{attribute 'GeneratedUsingTerminal: EL3773-0000-0016'}
{attribute addProperty BoxType "EL3773-0000-0016"}
{attribute addProperty Id "L1_Voltage_StatusAT %I*L1_Voltage_Status_784F03AD8L1_Voltage_SamplesAT %I*L1_Voltage_Samples_ED678DEE20L1_Current_SamplesAT %I*L1_Current_Samples_89E078188L1_Current_Samples_1AT %I*L1_Current_Samples_3209B12F20L2_Voltage_StatusAT %I*L2_Voltage_Status_0626A0108L2_Voltage_SamplesAT %I*L2_Voltage_Samples_D91109BE20L2_Current_StatusAT %I*L2_Current_Status_F789DBA58L2_Current_SamplesAT %I*L2_Current_Samples_067F357F20L3_Voltage_StatusAT %I*L3_Voltage_Status_2C01C17B8L3_Voltage_SamplesAT %I*L3_Voltage_Samples_CAC3758E20L3_Current_StatusAT %I*L3_Current_Status_DDAEBACE8L3_Current_SamplesAT %I*L3_Current_Samples_15AD494F20AI_Timestamp_NextSync1TimeAT %I*AI_Timestamp_NextSync1Time_9AFDC2758AI_CycleCountAT %I*AI_CycleCount_B1A935A22WcStateAT %I*WcState_9091E0EB2InfoDataAT %I*InfoData_1088C70510"}
{attribute addProperty CRC "1502544242"}
{attribute addProperty Size "190"}
TYPE EL3773_598F0172 EXTENDS EtcSlaveTerminalBase_947E5A46 :
STRUCT
	{attribute addProperty Name "L1_Voltage_Status"}
	L1_Voltage_Status : L1_Voltage_Status_784F03AD;
	{attribute addProperty Name "L1_Voltage_Samples"}
	L1_Voltage_Samples : L1_Voltage_Samples_ED678DEE;
	{attribute addProperty Name "L1_Current_Samples"}
	L1_Current_Samples : L1_Current_Samples_89E07818;
	{attribute addProperty Name "L1_Current_Samples_1"}
	L1_Current_Samples_1 : L1_Current_Samples_3209B12F;
	{attribute addProperty Name "L2_Voltage_Status"}
	L2_Voltage_Status : L2_Voltage_Status_0626A010;
	{attribute addProperty Name "L2_Voltage_Samples"}
	L2_Voltage_Samples : L2_Voltage_Samples_D91109BE;
	{attribute addProperty Name "L2_Current_Status"}
	L2_Current_Status : L2_Current_Status_F789DBA5;
	{attribute addProperty Name "L2_Current_Samples"}
	L2_Current_Samples : L2_Current_Samples_067F357F;
	{attribute addProperty Name "L3_Voltage_Status"}
	L3_Voltage_Status : L3_Voltage_Status_2C01C17B;
	{attribute addProperty Name "L3_Voltage_Samples"}
	L3_Voltage_Samples : L3_Voltage_Samples_CAC3758E;
	{attribute addProperty Name "L3_Current_Status"}
	L3_Current_Status : L3_Current_Status_DDAEBACE;
	{attribute addProperty Name "L3_Current_Samples"}
	L3_Current_Samples : L3_Current_Samples_15AD494F;
	{attribute addProperty Name "AI_Timestamp_NextSync1Time"}
	AI_Timestamp_NextSync1Time : AI_Timestamp_NextSync1Time_9AFDC275;
	{attribute addProperty Name "AI_CycleCount"}
	AI_CycleCount : AI_CycleCount_B1A935A2;
	{attribute addProperty Name "WcState"}
	WcState : WcState_9091E0EB;
	{attribute addProperty Name "InfoData"}
	InfoData : InfoData_1088C705;
END_STRUCT
END_TYPE

(* stored: Version 1.2.0.0, ProductVersion 3.1.4024.9
   DUT EL3773_598F0172: Id {b9d384b0-2ad7-4d38-8daf-73884c215fb2} *)
